FUNCTION_BLOCK _ETcVnBorderInterpolationMethod_TestSuite EXTENDS TcUnit.FB_TestSuite
VAR
END_VAR

TestAddress();
TestClearReference();
TestClone();
TestTypeNameReturnsExpected();
TestIdentifierReturnsExpected();
TestMakeReferenceToFollowsReference();
TestMakeReferenceToUpdatesReference();
TestSize();
TestValueReturnsExpectedAfterInit();
TestValueReturnsExpectedAfterChange();
TestSerializeTypeWith();
TestSerializeWith();
TestTryDeserializeFrom();
TestTryMakeReferenceToFollowsReference();
TestTryMakeReferenceToUpdatesReference();

METHOD PUBLIC TestAddress
VAR
    _type : _ETcVnBorderInterpolationMethod(ETcVnBorderInterpolationMethod.TCVN_BIM_CONSTANT);
    notExpected : PVOID := 0;
    actual : PVOID;
END_VAR
TEST('TestAddress');

actual := _type.Address;

AssertFalse(
    Condition := (notExpected = actual),
    Message := 'Type did not return a valid address.'
);

TEST_FINISHED();
END_METHOD

METHOD PUBLIC TestClearReference
VAR
    _type : _ETcVnBorderInterpolationMethod(ETcVnBorderInterpolationMethod.TCVN_BIM_CONSTANT);
	target : ETcVnBorderInterpolationMethod := ETcVnBorderInterpolationMethod.TCVN_BIM_CONSTANT;
    expected : ETcVnBorderInterpolationMethod := ETcVnBorderInterpolationMethod.TCVN_BIM_CONSTANT;
    actual : ETcVnBorderInterpolationMethod;
END_VAR
TEST('TestClearReference');

_type.MakeReferenceTo(target);
_type.ClearReference();
target := ETcVnBorderInterpolationMethod.TCVN_BIM_REPLICATE;

actual := _type.Value;

AssertEquals(
    Expected := expected,
    Actual := actual,
    Message := 'Value continued to follow target.'
);

TEST_FINISHED();
END_METHOD

METHOD PUBLIC TestClone
VAR
    _type : _ETcVnBorderInterpolationMethod(ETcVnBorderInterpolationMethod.TCVN_BIM_CONSTANT);
	clone : I_Datatype;
	isValidClone : BOOL;
	compareResult : DINT;
END_VAR
TEST('TestClone');

clone := _type.Clone();

isValidClone := clone <> 0;

IF isValidClone THEN
	compareResult := memcmp(_type.Address, clone.Address, clone.Size);
END_IF

AssertTrue(
	Condition := isValidClone,
	Message := 'Clone did not produce a clone'
);

AssertEquals_DINT(
	Expected := 0,
    Actual := compareResult,
    Message := 'Clone did not return a valid clone.'
);

clone.Dispose();

TEST_FINISHED();
END_METHOD

METHOD PUBLIC TestIdentifierReturnsExpected
VAR
    _type : _ETcVnBorderInterpolationMethod(ETcVnBorderInterpolationMethod.TCVN_BIM_CONSTANT);
    expected : STRING := 'ETcVnBorderInterpolationMethod';
    actual : STRING;
END_VAR
TEST('TestIdentifierReturnsExpected');

actual := _type.Identifier;

AssertEquals_STRING(
    Expected := expected,
    Actual := actual,
    Message := 'Type did not return correct iec type.'
);

TEST_FINISHED();
END_METHOD

METHOD PUBLIC TestMakeReferenceToFollowsReference
VAR
    _type : _ETcVnBorderInterpolationMethod(ETcVnBorderInterpolationMethod.TCVN_BIM_CONSTANT);
	target : ETcVnBorderInterpolationMethod := ETcVnBorderInterpolationMethod.TCVN_BIM_CONSTANT;
    expected : ETcVnBorderInterpolationMethod := ETcVnBorderInterpolationMethod.TCVN_BIM_REPLICATE;
    actual : ETcVnBorderInterpolationMethod;
END_VAR
TEST('TestMakeReferenceToFollowsReference');

_type.MakeReferenceTo(target);
target := ETcVnBorderInterpolationMethod.TCVN_BIM_REPLICATE;

actual := _type.Value;

AssertEquals(
    Expected := expected,
    Actual := actual,
    Message := 'Value did not follow target change.'
);

TEST_FINISHED();
END_METHOD

METHOD PUBLIC TestMakeReferenceToUpdatesReference
VAR
    _type : _ETcVnBorderInterpolationMethod(ETcVnBorderInterpolationMethod.TCVN_BIM_CONSTANT);
	target : ETcVnBorderInterpolationMethod := ETcVnBorderInterpolationMethod.TCVN_BIM_CONSTANT;
    expected : ETcVnBorderInterpolationMethod := ETcVnBorderInterpolationMethod.TCVN_BIM_REPLICATE;
    actual : ETcVnBorderInterpolationMethod;
END_VAR
TEST('TestMakeReferenceToUpdatesReference');

_type.MakeReferenceTo(target);
_type.Value := ETcVnBorderInterpolationMethod.TCVN_BIM_REPLICATE;

actual := target;

AssertEquals(
    Expected := expected,
    Actual := actual,
    Message := 'Value did not update target.'
);

TEST_FINISHED();
END_METHOD

METHOD PUBLIC TestSerializeTypeWith
VAR
    _type : _ETcVnBorderInterpolationMethod(ETcVnBorderInterpolationMethod.TCVN_BIM_CONSTANT);
    serializer : JsonSerializer;
    expected : STRING(500) := '{"typeName":"ENUM","identifier":"ETcVnBorderInterpolationMethod","enumerations":["TCVN_BIM_CONSTANT","TCVN_BIM_REPLICATE","TCVN_BIM_REFLECT","TCVN_BIM_WRAP","TCVN_BIM_REFLECT_101","TCVN_BIM_DEFAULT","TCVN_BIM_TRANSPARENT","TCVN_BIM_ISOLATED_CONSTANT","TCVN_BIM_ISOLATED_REPLICATE","TCVN_BIM_ISOLATED_REFLECT","TCVN_BIM_ISOLATED_WRAP","TCVN_BIM_ISOLATED_REFLECT_101"],"baseType":{"typeName":"DINT","minValue":-2147483648,"maxValue":2147483647,"isSigned":true,"isFloat":false}}'; 
    actual : STRING(500);
END_VAR
TEST('TestSerializeTypeWith');

serializer.Reset();
_type.SerializeTypeWith(serializer);
serializer.TryGetSerializedData(ADR(actual), SIZEOF(actual));

AssertEquals_STRING(
    Expected := expected,
    Actual := actual,
    Message := 'Serialization of type did not return correct string.'
);

TEST_FINISHED();
END_METHOD

METHOD PUBLIC TestSerializeWith
VAR
    _type : _ETcVnBorderInterpolationMethod(ETcVnBorderInterpolationMethod.TCVN_BIM_CONSTANT);
    serializer : JsonSerializer;
    expected : STRING := '"TCVN_BIM_CONSTANT"';
    actual : STRING(500);
END_VAR
TEST('TestSerializeWith');

serializer.Reset();
_type.SerializeWith(serializer);
serializer.TryGetSerializedData(ADR(actual), SIZEOF(actual));

AssertEquals_STRING(
    Expected := expected,
    Actual := actual,
    Message := 'Serialization of type data did not return correct string.'
);

TEST_FINISHED();
END_METHOD

METHOD PUBLIC TestSize
VAR
    _type : _ETcVnBorderInterpolationMethod(ETcVnBorderInterpolationMethod.TCVN_BIM_CONSTANT);
    expected : UDINT := SIZEOF(ETcVnBorderInterpolationMethod);
    actual : UDINT;
END_VAR
TEST('TestSize');

actual := _type.Size;

AssertEquals_UDINT(
    Expected := Expected,
    Actual := actual,
    Message := 'Type did not return the correct size.'
);

TEST_FINISHED();
END_METHOD

METHOD PUBLIC TestTryDeserializeFrom
VAR
    deserializer : JsonDeserializer;
    feedback : DeserializerFeedback;
    json : STRING := '"TCVN_BIM_CONSTANT"';
    _type : _ETcVnBorderInterpolationMethod(ETcVnBorderInterpolationMethod.TCVN_BIM_CONSTANT);
    expected : ETcVnBorderInterpolationMethod := ETcVnBorderInterpolationMethod.TCVN_BIM_CONSTANT;
    actual : ETcVnBorderInterpolationMethod;
 END_VAR
TEST('TestTryDeserializeFrom');

deserializer.Reset();
deserializer.TryLoad(json);
_type.TryDeserializeFrom(Deserializer, Feedback);

actual := _type.Value;

AssertEquals(
    Expected := expected,
    Actual := actual,
    Message := 'Type did not deserialize correctly.'
);

TEST_FINISHED();
END_METHOD

METHOD PUBLIC TestTryMakeReferenceToFollowsReference
VAR
    _type : _ETcVnBorderInterpolationMethod(ETcVnBorderInterpolationMethod.TCVN_BIM_CONSTANT);
	target : _ETcVnBorderInterpolationMethod(ETcVnBorderInterpolationMethod.TCVN_BIM_CONSTANT);
    expected : ETcVnBorderInterpolationMethod := ETcVnBorderInterpolationMethod.TCVN_BIM_REPLICATE;
    actual : ETcVnBorderInterpolationMethod;
END_VAR
TEST('TestTryMakeReferenceToFollowsReference');

_type.TryMakeReferenceTo(target);
target.Value := ETcVnBorderInterpolationMethod.TCVN_BIM_REPLICATE;

actual := _type.Value;

AssertEquals(
    Expected := expected,
    Actual := actual,
    Message := 'Value did not follow target change.'
);

TEST_FINISHED();
END_METHOD

METHOD PUBLIC TestTryMakeReferenceToUpdatesReference
VAR
    _type : _ETcVnBorderInterpolationMethod(ETcVnBorderInterpolationMethod.TCVN_BIM_CONSTANT);
	target : _ETcVnBorderInterpolationMethod(ETcVnBorderInterpolationMethod.TCVN_BIM_CONSTANT);
    expected : ETcVnBorderInterpolationMethod := ETcVnBorderInterpolationMethod.TCVN_BIM_REPLICATE;
    actual : ETcVnBorderInterpolationMethod;
END_VAR
TEST('TestTryMakeReferenceToUpdatesReference');

_type.TryMakeReferenceTo(target);
_type.Value := ETcVnBorderInterpolationMethod.TCVN_BIM_REPLICATE;

actual := target.Value;

AssertEquals(
    Expected := expected,
    Actual := actual,
    Message := 'Value did not update target.'
);

TEST_FINISHED();
END_METHOD

METHOD PUBLIC TestTypeNameReturnsExpected
VAR
    _type : _ETcVnBorderInterpolationMethod(ETcVnBorderInterpolationMethod.TCVN_BIM_CONSTANT);
    expected : STRING := 'ENUM';
    actual : STRING;
END_VAR
TEST('TestTypeNameReturnsExpected');

actual := _type.TypeName;

AssertEquals_STRING(
    Expected := expected,
    Actual := actual,
    Message := 'Type did not return correct iec type.'
);

TEST_FINISHED();
END_METHOD

METHOD PUBLIC TestValueReturnsExpectedAfterChange
VAR
    _type : _ETcVnBorderInterpolationMethod(ETcVnBorderInterpolationMethod.TCVN_BIM_CONSTANT);
    expected : ETcVnBorderInterpolationMethod := ETcVnBorderInterpolationMethod.TCVN_BIM_REPLICATE;
    actual : ETcVnBorderInterpolationMethod;
END_VAR
TEST('TestValueReturnsExpectedAfterChange');

_type.Value := ETcVnBorderInterpolationMethod.TCVN_BIM_REPLICATE;

actual := _type.Value;

AssertEquals(
    Expected := expected,
    Actual := actual,
    Message := 'Expected value not returned after change.'
);

TEST_FINISHED();
END_METHOD

METHOD PUBLIC TestValueReturnsExpectedAfterInit
VAR
    _type : _ETcVnBorderInterpolationMethod(ETcVnBorderInterpolationMethod.TCVN_BIM_CONSTANT);
    expected : ETcVnBorderInterpolationMethod := ETcVnBorderInterpolationMethod.TCVN_BIM_CONSTANT;
    actual : ETcVnBorderInterpolationMethod;
END_VAR
TEST('TestValueReturnsExpectedAfterInit');

actual := _type.Value;

AssertEquals(
    Expected := expected,
    Actual := actual,
    Message := 'Expected value not returned after Init.'
);

TEST_FINISHED();
END_METHOD

END_FUNCTION_BLOCK

(* stored: Version 1.1.0.1, ProductVersion 3.1.4024.12
   POU _ETcVnBorderInterpolationMethod_TestSuite: Id {5f35bc6c-f798-0649-07e2-dc47cd0a7720}, SpecialFunc None
   Method TestAddress: Id {0216a6b3-b635-03bc-1797-a087a7175d39}
   Method TestClearReference: Id {a304a14e-26bd-0c24-1667-58d604268348}
   Method TestClone: Id {fd511a45-28ef-0f7a-1ecc-c0bfd6092cfa}
   Method TestIdentifierReturnsExpected: Id {3ef40395-d4d1-0033-1701-2ff618fe6f6c}
   Method TestMakeReferenceToFollowsReference: Id {adf64dfe-2803-0019-0acb-3ff3fd426963}
   Method TestMakeReferenceToUpdatesReference: Id {061c261c-8dbc-0741-1238-aabebc8f6216}
   Method TestSerializeTypeWith: Id {a03d44ef-dd8b-0fb7-1bc2-fb228fb7e082}
   Method TestSerializeWith: Id {09462f73-90da-0d2c-12f7-47eb1b8a7c9d}
   Method TestSize: Id {c234b36d-20d7-0043-1918-3073ff27c56f}
   Method TestTryDeserializeFrom: Id {4c4d6d59-3d49-00a4-1939-983e501e61e5}
   Method TestTryMakeReferenceToFollowsReference: Id {ffeba741-7e05-0ae0-1359-feb98055783f}
   Method TestTryMakeReferenceToUpdatesReference: Id {a8f1fa02-2d62-071c-0685-0c7ad63d8247}
   Method TestTypeNameReturnsExpected: Id {fdbfeac6-6d94-0548-27ba-00aad3f5ffec}
   Method TestValueReturnsExpectedAfterChange: Id {1010f8f8-7d5e-04de-1623-93f3dd276236}
   Method TestValueReturnsExpectedAfterInit: Id {a4079a77-1e16-0e76-3ab5-4d49e27452b4} *)
